FUNCTION_BLOCK LowpassFilter
VAR_INPUT
	x : LREAL;
	y : LREAL;
	ydot : LREAL;
END_VAR
VAR_OUTPUT
	yout : LREAL;
	ydotout : LREAL;
END_VAR
VAR
	cutFreq : LREAL := 100.0;
	wcut: LREAL := 2 * pi * cutFreq;
	w: LREAL := 1/wcut;
	wwcut : LREAL := 1/w/w;
	dt_: LREAL:= 1.0/DINT_TO_LREAL(gvl.sampleRate);
	yddot: LREAL;
END_VAR

yddot := wwcut*(x - y - 2 * 0.707 * w * ydot);
ydotout := ydot + yddot * dt_;
yout := y + ydotout * dt_;

END_FUNCTION_BLOCK

(* stored: Version 1.1.0.1, ProductVersion 3.1.4024.2
   POU LowpassFilter: Id {be7d3aa7-8bde-449a-96dc-ee63b9d3bf3f}, SpecialFunc None *)
